(*********************************** G.D S.p.A. - Technical Department ***********************************
============= PROGRAM INFO ============
FOLDER:             TBD
MACHINES INVOLVED:  TBD 

============= DESCRIPTION =============
csp main interface program

============= REVISIONS ===============
Date		Version	 	Author      	Description             
----------	-------		------------  	--------------------------------------------
2019/09/27 	0000.00	 	M.Grasso		Creation of the PRG

**********************************************************************************************************)
PROGRAM _csp_case_transport_low
VAR
END_VAR

(* CSP *)
	(* TRANSPORT *)
		(* ACC-U-CHANGE *)
		csp_case_transport_accU_depth();
		csp_case_transport_accU_virtualMaster();
		(* LS *)
		(* OS *)
		csp_case_transport_os_minorPlow();
		(* TENSIONER *)
		;

END_PROGRAM

(* stored: Version 1.1.0.1, ProductVersion 3.1.4024.3
   POU _csp_case_transport_low: Id {19b1b664-3aab-4218-813d-221e1d398e8a}, SpecialFunc None *)
